{attribute 'linkalways'} 
{attribute 'no_explicit_call' := 'This FB is a CLASS and must be accessed using methods or properties'}
{attribute 'enable_dynamic_creation'}
FUNCTION_BLOCK _TcVnArray7_LREAL EXTENDS AliasDatatypeBase
VAR
	localData : TcVnArray7_LREAL;
	activeData : REFERENCE TO TcVnArray7_LREAL REF= localData;
	aliasBaseDatatype : _Array0to6OfLREAL;
END_VAR

PROPERTY PUBLIC Address : PVOID
GET
Address := ADR(activeData);
END_GET
END_PROPERTY

METHOD PUBLIC ClearReference
VAR_INPUT
END_VAR
activeData REF= localData;
SetBaseDatatypeReference();
END_METHOD

METHOD PUBLIC Clone : I_Datatype
VAR
    pClone : POINTER TO _TcVnArray7_LREAL;
END_VAR
pClone := __NEW(_TcVnArray7_LREAL);
Clone := pClone^;
END_METHOD

METHOD FB_init : BOOL
VAR_INPUT
	bInitRetains : BOOL; // if TRUE, the retain variables are initialized (warm start / cold start)
	bInCopyCode : BOOL;  // if TRUE, the instance afterwards gets moved into the copy code (online change)
	//InitialValue : TcVnArray7_LREAL; // if possible, not all values can be initialized
END_VAR
//localData := InitialValue; // if possible, not all values can be initialized
SetBaseDatatypeReference();
AddBaseDatatype(aliasBaseDatatype);
END_METHOD

PROPERTY PUBLIC Identifier : T_MAXSTRING
GET
Identifier := 'TcVnArray7_LREAL';
END_GET
END_PROPERTY

METHOD PUBLIC MakeReferenceTo
VAR_INPUT
	ReferenceTarget : REFERENCE TO TcVnArray7_LREAL;
END_VAR
activeData REF= ReferenceTarget;
SetBaseDatatypeReference();
END_METHOD

METHOD PROTECTED SetBaseDatatypeReference
VAR_INPUT
END_VAR
aliasBaseDatatype.MakeReferenceTo(activeData);
END_METHOD

PROPERTY PUBLIC Size : UDINT
GET
Size := SIZEOF(activeData);
END_GET
END_PROPERTY

METHOD TryMakeReferenceTo : BOOL
VAR_INPUT
	Target : I_Datatype;
END_VAR
VAR
	targetAsAlias : I_AliasDatatype;
	pTargetData : POINTER TO TcVnArray7_LREAL;
END_VAR
IF NOT Target.TryResolveAsAliasDatatype(targetAsAlias) THEN
	RETURN;
END_IF

IF targetAsAlias.Identifier <> Identifier THEN
	RETURN;
END_IF

pTargetData := Target.Address;
activeData REF= pTargetData^;
SetBaseDatatypeReference();
TryMakeReferenceTo := TRUE;
END_METHOD

PROPERTY PUBLIC Value : REFERENCE TO TcVnArray7_LREAL
GET
Value REF= activeData;
END_GET
END_PROPERTY

END_FUNCTION_BLOCK

(* stored: Version 1.1.0.1, ProductVersion 3.1.4024.13
   POU _TcVnArray7_LREAL: Id {04333e86-a522-0d29-385e-6d477d6a0bb6}, SpecialFunc None
   Folder Core: Id {45625f14-ed24-04f0-2537-5c05082ec197}
   Folder Protected: Id {74a82d8e-cda4-0e4b-36e0-12573aeed95d}
   Folder Customize: Id {70a9eca8-4d04-06b9-06b6-1d6ea480f6f4}
   Folder Constructor: Id {79f12c16-ac15-000d-2056-0ab568a0aef0}
   Property Address: Id {c6000114-026b-0fdd-3d61-d41833895cf5}
   Get Get: Id {fdcd4517-a5bd-0a9b-1bfe-5f41090ead29}
   Method ClearReference: Id {feca4a44-bd99-0fcd-14d9-e3eeabe90c87}
   Method Clone: Id {ac0b14b0-70d0-08ed-2ac2-0ef1d4c9c808}
   Method FB_init: Id {832189c4-752b-061c-3290-e55403ec8c5a}
   Property Identifier: Id {9efcf5b5-aef3-0c11-3620-850771d79481}
   Get Get: Id {a916fbcc-6d6a-0356-111e-2e1d29522865}
   Method MakeReferenceTo: Id {c1701d7e-3689-0cef-234e-a213a172398c}
   Method SetBaseDatatypeReference: Id {ecae7616-57d3-0e1c-1d99-e2b92773c813}
   Property Size: Id {506b30e4-5926-09f0-2c79-1d23cc62d8cf}
   Get Get: Id {6eb2b044-cb39-0e57-1404-ffe86b63bee1}
   Method TryMakeReferenceTo: Id {13452747-8d59-081d-023f-9325eeb1b42f}
   Property Value: Id {0b1f69bb-c4ac-07ba-0de1-311f7ef59fb7}
   Get Get: Id {a1e37f84-1d8f-03ca-335c-629acec8e09b} *)
